DATA_BLOCK "DB104"
{ S7_Optimized_Access := 'FALSE' }
VERSION : 0.1
NON_RETAIN
   VAR
      DB104_DBD0 : Real;
      DB104_DBD4 : Real;
      DB104_DBD8 : Real;
      DB104_DBD12 : Real;
      DB104_DBD16 : Real;
      DB104_DBD20 : Real;
      DB104_DBD24 : Real;
      DB104_DBD28 : Real;
      DB104_DBD32 : Real;
      DB104_DBD36 : Real;
      DB104_DBD40 : Real;
      DB104_DBD44 : Real;
      DB104_DBD48 : Real;
      DB104_DBD52 : Real;
      DB104_DBD56 : Real;
      DB104_DBD60 : Real;
      DB104_DBD64 : Real;
      DB104_DBD68 : Real;
      DB104_DBD72 : Real;
      DB104_DBD76 : Real;
      DB104_DBD80 : Real;
      DB104_DBD84 : Real;
      DB104_DBD88 : Real;
      DB104_DBD92 : Real;
      DB104_DBD96 : Real;
      DB104_DBD100 : Real;
      DB104_DBD104 : Real;
      DB104_DBD108 : Real;
      DB104_DBD112 : Real;
      DB104_DBD116 : Real;
      DB104_DBD120 : Real;
      DB104_DBD124 : Real;
      DB104_DBD128 : Real;
      DB104_DBD132 : Real;
      DB104_DBD136 : Real;
      DB104_DBD140 : Real;
      DB104_DBD144 : Real;
      DB104_DBD148 : Real;
      DB104_DBD152 : Real;
      DB104_DBD156 : Real;
      DB104_DBD160 : Real;
      DB104_DBD164 : Real;
      DB104_DBD168 : Real;
      DB104_DBD172 : Real;
      DB104_DBD176 : Real;
      DB104_DBD180 : Real;
      DB104_DBD184 : Real;
      DB104_DBD188 : Real;
      DB104_DBD192 : Real;
      DB104_DBD196 : Real;
      DB104_DBD200 : Real;
      DB104_DBD204 : Real;
      DB104_DBD208 : Real;
      DB104_DBD212 : Real;
      DB104_DBD216 : Real;
      DB104_DBD220 : Real;
      DB104_DBD224 : Real;
      DB104_DBD228 : Real;
      DB104_DBD232 : Real;
      DB104_DBD236 : Real;
      DB104_DBD240 : Real;
      DB104_DBD244 : Real;
      DB104_DBD248 : Real;
      DB104_DBD252 : Real;
      DB104_DBD256 : Real;
      DB104_DBD260 : Real;
      DB104_DBD264 : Real;
      DB104_DBD268 : Real;
      DB104_DBD272 : Real;
      DB104_DBD276 : Real;
      DB104_DBD280 : Real;
      DB104_DBD284 : Real;
      DB104_DBD288 : Real;
      DB104_DBD292 : Real;
      DB104_DBD296 : Real;
      DB104_DBD300 : Real;
      DB104_DBD304 : Real;
      DB104_DBD308 : Real;
      DB104_DBD312 : Real;
      DB104_DBD316 : Real;
      DB104_DBD800 : Real;
      DB104_DBD804 : Real;
      DB104_DBD808 : Real;
      DB104_DBD812 : Real;
      DB104_DBD816 : Real;
      DB104_DBD820 : Real;
      DB104_DBD824 : Real;
      DB104_DBD828 : Real;
      DB104_DBD832 : Real;
      DB104_DBD836 : Real;
      DB104_DBD840 : Real;
      DB104_DBD844 : Real;
      DB104_DBD848 : Real;
      DB104_DBD852 : Real;
      DB104_DBD856 : Real;
      DB104_DBD860 : Real;
      DB104_DBD864 : Real;
      DB104_DBD868 : Real;
      DB104_DBD872 : Real;
      DB104_DBD876 : Real;
      DB104_DBD880 : Real;
      DB104_DBD884 : Real;
      DB104_DBD888 : Real;
      DB104_DBD892 : Real;
      DB104_DBD896 : Real;
      DB104_DBD900 : Real;
      DB104_DBD904 : Real;
      DB104_DBD908 : Real;
      DB104_DBD912 : Real;
      DB104_DBD916 : Real;
      DB104_DBD920 : Real;
      DB104_DBD924 : Real;
      DB104_DBD928 : Real;
      DB104_DBD932 : Real;
      DB104_DBD936 : Real;
      DB104_DBD940 : Real;
      DB104_DBD944 : Real;
      DB104_DBD948 : Real;
      DB104_DBD952 : Real;
      DB104_DBD956 : Real;
      DB104_DBD960 : Real;
      DB104_DBD964 : Real;
      DB104_DBD968 : Real;
      DB104_DBD972 : Real;
      DB104_DBD976 : Real;
      DB104_DBD980 : Real;
      DB104_DBD984 : Real;
      DB104_DBD988 : Real;
      DB104_DBD992 : Real;
      DB104_DBD996 : Real;
      DB104_DBD1000 : Real;
      DB104_DBD1004 : Real;
      DB104_DBD1008 : Real;
      DB104_DBD1012 : Real;
      DB104_DBD1016 : Real;
      DB104_DBD1020 : Real;
      DB104_DBD1024 : Real;
      DB104_DBD1028 : Real;
      DB104_DBD1032 : Real;
      DB104_DBD1036 : Real;
      DB104_DBD1040 : Real;
      DB104_DBD1044 : Real;
      DB104_DBD1048 : Real;
      DB104_DBD1052 : Real;
      DB104_DBD1056 : Real;
      DB104_DBD1060 : Real;
      DB104_DBD1064 : Real;
      DB104_DBD1068 : Real;
      DB104_DBD1072 : Real;
      DB104_DBD1076 : Real;
      DB104_DBD1080 : Real;
      DB104_DBD1084 : Real;
      DB104_DBD1088 : Real;
      DB104_DBD1092 : Real;
      DB104_DBD1096 : Real;
      DB104_DBD1100 : Real;
      DB104_DBD1104 : Real;
      DB104_DBD1108 : Real;
      DB104_DBD1112 : Real;
      DB104_DBD1116 : Real;
      DB104_DBD1600 : Real;
      DB104_DBD1604 : Real;
      DB104_DBD1608 : Real;
      DB104_DBD1612 : Real;
      DB104_DBD1616 : Real;
      DB104_DBD1620 : Real;
      DB104_DBD1624 : Real;
      DB104_DBD1628 : Real;
      DB104_DBD1632 : Real;
      DB104_DBD1636 : Real;
      DB104_DBD1640 : Real;
      DB104_DBD1644 : Real;
      DB104_DBD1648 : Real;
      DB104_DBD1652 : Real;
      DB104_DBD1656 : Real;
      DB104_DBD1660 : Real;
      DB104_DBD1664 : Real;
      DB104_DBD1668 : Real;
      DB104_DBD1672 : Real;
      DB104_DBD1676 : Real;
      DB104_DBD1680 : Real;
      DB104_DBD1684 : Real;
      DB104_DBD1688 : Real;
      DB104_DBD1692 : Real;
      DB104_DBD1696 : Real;
      DB104_DBD1700 : Real;
      DB104_DBD1704 : Real;
      DB104_DBD1708 : Real;
      DB104_DBD1712 : Real;
      DB104_DBD1716 : Real;
      DB104_DBD1720 : Real;
      DB104_DBD1724 : Real;
      DB104_DBD1728 : Real;
      DB104_DBD1732 : Real;
      DB104_DBD1736 : Real;
      DB104_DBD1740 : Real;
      DB104_DBD1744 : Real;
      DB104_DBD1748 : Real;
      DB104_DBD1752 : Real;
      DB104_DBD1756 : Real;
      DB104_DBD1760 : Real;
      DB104_DBD1764 : Real;
      DB104_DBD1768 : Real;
      DB104_DBD1772 : Real;
      DB104_DBD1776 : Real;
      DB104_DBD1780 : Real;
      DB104_DBD1784 : Real;
      DB104_DBD1788 : Real;
      DB104_DBD1792 : Real;
      DB104_DBD1796 : Real;
      DB104_DBD1800 : Real;
      DB104_DBD1804 : Real;
      DB104_DBD1808 : Real;
      DB104_DBD1812 : Real;
      DB104_DBD1816 : Real;
      DB104_DBD1820 : Real;
      DB104_DBD1824 : Real;
      DB104_DBD1828 : Real;
      DB104_DBD1832 : Real;
      DB104_DBD1836 : Real;
      DB104_DBD1840 : Real;
      DB104_DBD1844 : Real;
      DB104_DBD1848 : Real;
      DB104_DBD1852 : Real;
      DB104_DBD1856 : Real;
      DB104_DBD1860 : Real;
      DB104_DBD1864 : Real;
      DB104_DBD1868 : Real;
      DB104_DBD1872 : Real;
      DB104_DBD1876 : Real;
      DB104_DBD1880 : Real;
      DB104_DBD1884 : Real;
      DB104_DBD1888 : Real;
      DB104_DBD1892 : Real;
      DB104_DBD1896 : Real;
      DB104_DBD1900 : Real;
      DB104_DBD1904 : Real;
      DB104_DBD1908 : Real;
      DB104_DBD1912 : Real;
      DB104_DBD1916 : Real;
      DB104_DBD2400 : Real;
      DB104_DBD2404 : Real;
      DB104_DBD2408 : Real;
      DB104_DBD2412 : Real;
      DB104_DBD2416 : Real;
      DB104_DBD2420 : Real;
      DB104_DBD2424 : Real;
      DB104_DBD2428 : Real;
      DB104_DBD2432 : Real;
      DB104_DBD2436 : Real;
      DB104_DBD2440 : Real;
      DB104_DBD2444 : Real;
      DB104_DBD2448 : Real;
      DB104_DBD2452 : Real;
      DB104_DBD2456 : Real;
      DB104_DBD2460 : Real;
      DB104_DBD2464 : Real;
      DB104_DBD2468 : Real;
      DB104_DBD2472 : Real;
      DB104_DBD2476 : Real;
      DB104_DBD2480 : Real;
      DB104_DBD2484 : Real;
      DB104_DBD2488 : Real;
      DB104_DBD2492 : Real;
      DB104_DBD2496 : Real;
      DB104_DBD2500 : Real;
      DB104_DBD2504 : Real;
      DB104_DBD2508 : Real;
      DB104_DBD2512 : Real;
      DB104_DBD2516 : Real;
      DB104_DBD2520 : Real;
      DB104_DBD2524 : Real;
      DB104_DBD2528 : Real;
      DB104_DBD2532 : Real;
      DB104_DBD2536 : Real;
      DB104_DBD2540 : Real;
      DB104_DBD2544 : Real;
      DB104_DBD2548 : Real;
      DB104_DBD2552 : Real;
      DB104_DBD2556 : Real;
      DB104_DBD2560 : Real;
      DB104_DBD2564 : Real;
      DB104_DBD2568 : Real;
      DB104_DBD2572 : Real;
      DB104_DBD2576 : Real;
      DB104_DBD2580 : Real;
      DB104_DBD2584 : Real;
      DB104_DBD2588 : Real;
      DB104_DBD2592 : Real;
      DB104_DBD2596 : Real;
      DB104_DBD2600 : Real;
      DB104_DBD2604 : Real;
      DB104_DBD2608 : Real;
      DB104_DBD2612 : Real;
      DB104_DBD2616 : Real;
      DB104_DBD2620 : Real;
      DB104_DBD2624 : Real;
      DB104_DBD2628 : Real;
      DB104_DBD2632 : Real;
      DB104_DBD2636 : Real;
      DB104_DBD2640 : Real;
      DB104_DBD2644 : Real;
      DB104_DBD2648 : Real;
      DB104_DBD2652 : Real;
      DB104_DBD2656 : Real;
      DB104_DBD2660 : Real;
      DB104_DBD2664 : Real;
      DB104_DBD2668 : Real;
      DB104_DBD2672 : Real;
      DB104_DBD2676 : Real;
      DB104_DBD2680 : Real;
      DB104_DBD2684 : Real;
      DB104_DBD2688 : Real;
      DB104_DBD2692 : Real;
      DB104_DBD2696 : Real;
      DB104_DBD2700 : Real;
      DB104_DBD2704 : Real;
      DB104_DBD2708 : Real;
      DB104_DBD2712 : Real;
      DB104_DBD2716 : Real;
   END_VAR


BEGIN

END_DATA_BLOCK

DATA_BLOCK "DB101"
{ S7_Optimized_Access := 'FALSE' }
VERSION : 0.1
NON_RETAIN
   VAR
      DB101_DBW0 : Word;
      DB101_DBW2 : Word;
      DB101_DBD4 : Real;
      DB101_DBD8 : Real;
      DB101_DBD12 : Real;
      DB101_DBD16 : Real;
      DB101_DBD96 : Real;
      DB101_DBW176 : Word;
      DB101_DBW178 : Word;
      DB101_DBW180 : Word;
      DB101_DBW182 : Word;
      DB101_DBW184 : Word;
      DB101_DBW186 : Word;
      DB101_DBW188 : Word;
      DB101_DBW190 : Word;
      DB101_DBW192 : Word;
      DB101_DBW194 : Word;
      DB101_DBW196 : Word;
      DB101_DBW198 : Word;
      DB101_DBW200 : Word;
      DB101_DBW202 : Word;
      DB101_DBW204 : Word;
      DB101_DBW206 : Word;
      DB101_DBW208 : Word;
      DB101_DBW210 : Word;
      DB101_DBW212 : Word;
      DB101_DBW214 : Word;
      DB101_DBW216 : Word;
      DB101_DBW218 : Word;
      DB101_DBW220 : Word;
      DB101_DBW222 : Word;
      DB101_DBW224 : Word;
      DB101_DBW226 : Word;
      DB101_DBW228 : Word;
      DB101_DBW230 : Word;
      DB101_DBW232 : Word;
      DB101_DBW234 : Word;
      DB101_DBW236 : Word;
      DB101_DBW238 : Word;
      DB101_DBW240 : Word;
      DB101_DBW242 : Word;
      DB101_DBW244 : Word;
      DB101_DBW246 : Word;
      DB101_DBW248 : Word;
      DB101_DBW250 : Word;
      DB101_DBW252 : Word;
      DB101_DBW254 : Word;
      DB101_DBW256 : Word;
      DB101_DBW258 : Word;
      DB101_DBW260 : Word;
      DB101_DBW262 : Word;
      DB101_DBW264 : Word;
      DB101_DBW266 : Word;
      DB101_DBW268 : Word;
      DB101_DBW270 : Word;
      DB101_DBW272 : Word;
      DB101_DBW274 : Word;
      DB101_DBW276 : Word;
      DB101_DBW278 : Word;
      DB101_DBW280 : Word;
      DB101_DBW282 : Word;
      DB101_DBW284 : Word;
      DB101_DBW286 : Word;
      DB101_DBW288 : Word;
      DB101_DBW290 : Word;
      DB101_DBW292 : Word;
      DB101_DBW294 : Word;
      DB101_DBW296 : Word;
      DB101_DBW298 : Word;
      DB101_DBW300 : Word;
      DB101_DBW302 : Word;
      DB101_DBW304 : Word;
      DB101_DBW306 : Word;
      DB101_DBW308 : Word;
      DB101_DBW310 : Word;
      DB101_DBW312 : Word;
      DB101_DBW314 : Word;
      DB101_DBW316 : Word;
      DB101_DBW318 : Word;
      DB101_DBW320 : Word;
      DB101_DBW322 : Word;
      DB101_DBW324 : Word;
      DB101_DBW326 : Word;
      DB101_DBW328 : Word;
      DB101_DBW330 : Word;
      DB101_DBW332 : Word;
      DB101_DBW334 : Word;
      DB101_DBW576 : Word;
      DB101_DBW578 : Word;
      DB101_DBW580 : Word;
      DB101_DBW582 : Word;
      DB101_DBW584 : Word;
      DB101_DBW586 : Word;
      DB101_DBW588 : Word;
      DB101_DBW590 : Word;
      DB101_DBW592 : Word;
      DB101_DBW594 : Word;
      DB101_DBW596 : Word;
      DB101_DBW598 : Word;
      DB101_DBW600 : Word;
      DB101_DBW602 : Word;
      DB101_DBW604 : Word;
      DB101_DBW606 : Word;
      DB101_DBW608 : Word;
      DB101_DBW610 : Word;
      DB101_DBW612 : Word;
      DB101_DBW614 : Word;
      DB101_DBW616 : Word;
      DB101_DBW618 : Word;
      DB101_DBW620 : Word;
      DB101_DBW622 : Word;
      DB101_DBW624 : Word;
      DB101_DBW626 : Word;
      DB101_DBW628 : Word;
      DB101_DBW630 : Word;
      DB101_DBW632 : Word;
      DB101_DBW634 : Word;
      DB101_DBW636 : Word;
      DB101_DBW638 : Word;
      DB101_DBW640 : Word;
      DB101_DBW642 : Word;
      DB101_DBW644 : Word;
      DB101_DBW646 : Word;
      DB101_DBW648 : Word;
      DB101_DBW650 : Word;
      DB101_DBW652 : Word;
      DB101_DBW654 : Word;
      DB101_DBW656 : Word;
      DB101_DBW658 : Word;
      DB101_DBW660 : Word;
      DB101_DBW662 : Word;
      DB101_DBW664 : Word;
      DB101_DBW666 : Word;
      DB101_DBW668 : Word;
      DB101_DBW670 : Word;
      DB101_DBW672 : Word;
      DB101_DBW674 : Word;
      DB101_DBW676 : Word;
      DB101_DBW678 : Word;
      DB101_DBW680 : Word;
      DB101_DBW682 : Word;
      DB101_DBW684 : Word;
      DB101_DBW686 : Word;
      DB101_DBW688 : Word;
      DB101_DBW690 : Word;
      DB101_DBW692 : Word;
      DB101_DBW694 : Word;
      DB101_DBW696 : Word;
      DB101_DBW698 : Word;
      DB101_DBW700 : Word;
      DB101_DBW702 : Word;
      DB101_DBW704 : Word;
      DB101_DBW706 : Word;
      DB101_DBW708 : Word;
      DB101_DBW710 : Word;
      DB101_DBW712 : Word;
      DB101_DBW714 : Word;
      DB101_DBW716 : Word;
      DB101_DBW718 : Word;
      DB101_DBW720 : Word;
      DB101_DBW722 : Word;
      DB101_DBW724 : Word;
      DB101_DBW726 : Word;
      DB101_DBW728 : Word;
      DB101_DBW730 : Word;
      DB101_DBW732 : Word;
      DB101_DBW734 : Word;
      DB101_DBW976 : Word;
      DB101_DBW978 : Word;
      DB101_DBW980 : Word;
      DB101_DBW982 : Word;
      DB101_DBW984 : Word;
      DB101_DBW986 : Word;
      DB101_DBW988 : Word;
      DB101_DBW990 : Word;
      DB101_DBW992 : Word;
      DB101_DBW994 : Word;
      DB101_DBW1016 : Word;
      DB101_DBW1018 : Word;
      DB101_DBW1020 : Word;
      DB101_DBW1022 : Word;
      DB101_DBW1024 : Word;
      DB101_DBW1026 : Word;
      DB101_DBW1028 : Word;
      DB101_DBW1030 : Word;
      DB101_DBW1032 : Word;
      DB101_DBW1034 : Word;
      DB101_DBW1056 : Word;
      DB101_DBW1058 : Word;
      DB101_DBW1060 : Word;
      DB101_DBW1062 : Word;
      DB101_DBW1064 : Word;
      DB101_DBW1066 : Word;
      DB101_DBW1068 : Word;
      DB101_DBW1070 : Word;
      DB101_DBW1072 : Word;
      DB101_DBW1074 : Word;
      DB101_DBW1096 : Word;
      DB101_DBW1098 : Word;
      DB101_DBW1100 : Word;
      DB101_DBW1102 : Word;
      DB101_DBW1104 : Word;
      DB101_DBW1106 : Word;
      DB101_DBW1108 : Word;
      DB101_DBW1110 : Word;
      DB101_DBW1112 : Word;
      DB101_DBW1114 : Word;
      DB101_DBX1136_0 : Bool;
      DB101_DBX1136_1 : Bool;
      DB101_DBX1136_2 : Bool;
      DB101_DBX1136_3 : Bool;
      DB101_DBX1136_4 : Bool;
      DB101_DBX1136_5 : Bool;
      DB101_DBX1136_6 : Bool;
      DB101_DBX1136_7 : Bool;
      DB101_DBX1137_0 : Bool;
      DB101_DBX1137_1 : Bool;
      DB101_DBX1140_0 : Bool;
      DB101_DBX1140_1 : Bool;
      DB101_DBX1140_2 : Bool;
      DB101_DBX1140_3 : Bool;
      DB101_DBX1140_4 : Bool;
      DB101_DBX1140_5 : Bool;
      DB101_DBX1140_6 : Bool;
      DB101_DBX1140_7 : Bool;
      DB101_DBX1141_0 : Bool;
      DB101_DBX1141_1 : Bool;
      DB101_DBD1144 : Real;
      DB101_DBD1224 : Real;
      DB101_DBW1304 : Word;
      DB101_DBW1306 : Word;
      DB101_DBW1308 : Word;
      DB101_DBW1310 : Word;
      DB101_DBW1312 : Word;
      DB101_DBW1314 : Word;
      DB101_DBW1316 : Word;
      DB101_DBW1318 : Word;
      DB101_DBW1320 : Word;
      DB101_DBW1322 : Word;
      DB101_DBW1324 : Word;
      DB101_DBW1326 : Word;
      DB101_DBW1328 : Word;
      DB101_DBW1330 : Word;
      DB101_DBW1332 : Word;
      DB101_DBW1334 : Word;
      DB101_DBW1336 : Word;
      DB101_DBW1338 : Word;
      DB101_DBW1340 : Word;
      DB101_DBW1342 : Word;
      DB101_DBW1344 : Word;
      DB101_DBW1346 : Word;
      DB101_DBW1348 : Word;
      DB101_DBW1350 : Word;
      DB101_DBW1352 : Word;
      DB101_DBW1354 : Word;
      DB101_DBW1356 : Word;
      DB101_DBW1358 : Word;
      DB101_DBW1360 : Word;
      DB101_DBW1362 : Word;
      DB101_DBW1364 : Word;
      DB101_DBW1366 : Word;
      DB101_DBW1368 : Word;
      DB101_DBW1370 : Word;
      DB101_DBW1372 : Word;
      DB101_DBW1374 : Word;
      DB101_DBW1376 : Word;
      DB101_DBW1378 : Word;
      DB101_DBW1380 : Word;
      DB101_DBW1382 : Word;
      DB101_DBW1384 : Word;
      DB101_DBW1386 : Word;
      DB101_DBW1388 : Word;
      DB101_DBW1390 : Word;
      DB101_DBW1392 : Word;
      DB101_DBW1394 : Word;
      DB101_DBW1396 : Word;
      DB101_DBW1398 : Word;
      DB101_DBW1400 : Word;
      DB101_DBW1402 : Word;
      DB101_DBW1404 : Word;
      DB101_DBW1406 : Word;
      DB101_DBW1408 : Word;
      DB101_DBW1410 : Word;
      DB101_DBW1412 : Word;
      DB101_DBW1414 : Word;
      DB101_DBW1416 : Word;
      DB101_DBW1418 : Word;
      DB101_DBW1420 : Word;
      DB101_DBW1422 : Word;
      DB101_DBW1424 : Word;
      DB101_DBW1426 : Word;
      DB101_DBW1428 : Word;
      DB101_DBW1430 : Word;
      DB101_DBW1432 : Word;
      DB101_DBW1434 : Word;
      DB101_DBW1436 : Word;
      DB101_DBW1438 : Word;
      DB101_DBW1440 : Word;
      DB101_DBW1442 : Word;
      DB101_DBW1444 : Word;
      DB101_DBW1446 : Word;
      DB101_DBW1448 : Word;
      DB101_DBW1450 : Word;
      DB101_DBW1452 : Word;
      DB101_DBW1454 : Word;
      DB101_DBW1456 : Word;
      DB101_DBW1458 : Word;
      DB101_DBW1460 : Word;
      DB101_DBW1462 : Word;
      DB101_DBW1704 : Word;
      DB101_DBW1706 : Word;
      DB101_DBW1708 : Word;
      DB101_DBW1710 : Word;
      DB101_DBW1712 : Word;
      DB101_DBW1714 : Word;
      DB101_DBW1716 : Word;
      DB101_DBW1718 : Word;
      DB101_DBW1720 : Word;
      DB101_DBW1722 : Word;
      DB101_DBW1724 : Word;
      DB101_DBW1726 : Word;
      DB101_DBW1728 : Word;
      DB101_DBW1730 : Word;
      DB101_DBW1732 : Word;
      DB101_DBW1734 : Word;
      DB101_DBW1736 : Word;
      DB101_DBW1738 : Word;
      DB101_DBW1740 : Word;
      DB101_DBW1742 : Word;
      DB101_DBW1744 : Word;
      DB101_DBW1746 : Word;
      DB101_DBW1748 : Word;
      DB101_DBW1750 : Word;
      DB101_DBW1752 : Word;
      DB101_DBW1754 : Word;
      DB101_DBW1756 : Word;
      DB101_DBW1758 : Word;
      DB101_DBW1760 : Word;
      DB101_DBW1762 : Word;
      DB101_DBW1764 : Word;
      DB101_DBW1766 : Word;
      DB101_DBW1768 : Word;
      DB101_DBW1770 : Word;
      DB101_DBW1772 : Word;
      DB101_DBW1774 : Word;
      DB101_DBW1776 : Word;
      DB101_DBW1778 : Word;
      DB101_DBW1780 : Word;
      DB101_DBW1782 : Word;
      DB101_DBW1784 : Word;
      DB101_DBW1786 : Word;
      DB101_DBW1788 : Word;
      DB101_DBW1790 : Word;
      DB101_DBW1792 : Word;
      DB101_DBW1794 : Word;
      DB101_DBW1796 : Word;
      DB101_DBW1798 : Word;
      DB101_DBW1800 : Word;
      DB101_DBW1802 : Word;
      DB101_DBW1804 : Word;
      DB101_DBW1806 : Word;
      DB101_DBW1808 : Word;
      DB101_DBW1810 : Word;
      DB101_DBW1812 : Word;
      DB101_DBW1814 : Word;
      DB101_DBW1816 : Word;
      DB101_DBW1818 : Word;
      DB101_DBW1820 : Word;
      DB101_DBW1822 : Word;
      DB101_DBW1824 : Word;
      DB101_DBW1826 : Word;
      DB101_DBW1828 : Word;
      DB101_DBW1830 : Word;
      DB101_DBW1832 : Word;
      DB101_DBW1834 : Word;
      DB101_DBW1836 : Word;
      DB101_DBW1838 : Word;
      DB101_DBW1840 : Word;
      DB101_DBW1842 : Word;
      DB101_DBW1844 : Word;
      DB101_DBW1846 : Word;
      DB101_DBW1848 : Word;
      DB101_DBW1850 : Word;
      DB101_DBW1852 : Word;
      DB101_DBW1854 : Word;
      DB101_DBW1856 : Word;
      DB101_DBW1858 : Word;
      DB101_DBW1860 : Word;
      DB101_DBW1862 : Word;
      DB101_DBW2104 : Word;
      DB101_DBW2106 : Word;
      DB101_DBW2108 : Word;
      DB101_DBW2110 : Word;
      DB101_DBW2112 : Word;
      DB101_DBW2114 : Word;
      DB101_DBW2116 : Word;
      DB101_DBW2118 : Word;
      DB101_DBW2120 : Word;
      DB101_DBW2122 : Word;
      DB101_DBW2144 : Word;
      DB101_DBW2146 : Word;
      DB101_DBW2148 : Word;
      DB101_DBW2150 : Word;
      DB101_DBW2152 : Word;
      DB101_DBW2154 : Word;
      DB101_DBW2156 : Word;
      DB101_DBW2158 : Word;
      DB101_DBW2160 : Word;
      DB101_DBW2162 : Word;
      DB101_DBW2184 : Word;
      DB101_DBW2186 : Word;
      DB101_DBW2188 : Word;
      DB101_DBW2190 : Word;
      DB101_DBW2192 : Word;
      DB101_DBW2194 : Word;
      DB101_DBW2196 : Word;
      DB101_DBW2198 : Word;
      DB101_DBW2200 : Word;
      DB101_DBW2202 : Word;
      DB101_DBW2224 : Word;
      DB101_DBW2226 : Word;
      DB101_DBW2228 : Word;
      DB101_DBW2230 : Word;
      DB101_DBW2232 : Word;
      DB101_DBW2234 : Word;
      DB101_DBW2236 : Word;
      DB101_DBW2238 : Word;
      DB101_DBW2240 : Word;
      DB101_DBW2242 : Word;
      DB101_DBX2264_0 : Bool;
      DB101_DBX2264_1 : Bool;
      DB101_DBX2264_2 : Bool;
      DB101_DBX2264_3 : Bool;
      DB101_DBX2264_4 : Bool;
      DB101_DBX2264_5 : Bool;
      DB101_DBX2264_6 : Bool;
      DB101_DBX2264_7 : Bool;
      DB101_DBX2265_0 : Bool;
      DB101_DBX2265_1 : Bool;
      DB101_DBX2268_0 : Bool;
      DB101_DBX2268_1 : Bool;
      DB101_DBX2268_2 : Bool;
      DB101_DBX2268_3 : Bool;
      DB101_DBX2268_4 : Bool;
      DB101_DBX2268_5 : Bool;
      DB101_DBX2268_6 : Bool;
      DB101_DBX2268_7 : Bool;
      DB101_DBX2269_0 : Bool;
      DB101_DBX2269_1 : Bool;
      DB101_DBW2272 : Word;
      DB101_DBW2274 : Word;
      DB101_DBD2276 : Real;
      DB101_DBD2280 : Real;
      DB101_DBD2284 : Real;
      DB101_DBD2288 : Real;
      DB101_DBD2292 : Real;
      DB101_DBD2296 : Real;
      DB101_DBD2300 : Real;
      DB101_DBD2304 : Real;
      DB101_DBD2308 : Real;
      DB101_DBD2312 : Real;
      DB101_DBD2316 : Real;
      DB101_DBD2320 : Real;
      DB101_DBD2324 : Real;
      DB101_DBD2328 : Real;
      DB101_DBD2332 : Real;
      DB101_DBD2336 : Real;
      DB101_DBD2340 : Real;
      DB101_DBD2344 : Real;
      DB101_DBD2348 : Real;
      DB101_DBD2352 : Real;
      DB101_DBD2356 : Real;
      DB101_DBD2360 : Real;
      DB101_DBD2364 : Real;
      DB101_DBD2368 : Real;
      DB101_DBD2372 : Real;
      DB101_DBD2376 : Real;
      DB101_DBD2380 : Real;
      DB101_DBD2384 : Real;
      DB101_DBD2388 : Real;
      DB101_DBD2392 : Real;
      DB101_DBD2676 : Real;
      DB101_DBD2680 : Real;
      DB101_DBD2684 : Real;
      DB101_DBD2688 : Real;
      DB101_DBD2692 : Real;
      DB101_DBD2696 : Real;
      DB101_DBD2700 : Real;
      DB101_DBD2704 : Real;
      DB101_DBD2708 : Real;
      DB101_DBD2712 : Real;
      DB101_DBD2716 : Real;
      DB101_DBD2720 : Real;
      DB101_DBD2724 : Real;
      DB101_DBD2728 : Real;
      DB101_DBD2732 : Real;
      DB101_DBD2736 : Real;
      DB101_DBD2740 : Real;
      DB101_DBD2744 : Real;
      DB101_DBD2748 : Real;
      DB101_DBD2752 : Real;
      DB101_DBD2756 : Real;
      DB101_DBD2760 : Real;
      DB101_DBD2764 : Real;
      DB101_DBD2768 : Real;
      DB101_DBD2772 : Real;
      DB101_DBD2776 : Real;
      DB101_DBD2780 : Real;
      DB101_DBD2784 : Real;
      DB101_DBD2788 : Real;
      DB101_DBD2792 : Real;
      DB101_DBD3076 : Real;
      DB101_DBD3080 : Real;
      DB101_DBW3086 : Word;
      DB101_DBW3088 : Word;
      DB101_DBD3090 : Real;
      DB101_DBD3094 : Real;
      DB101_DBW3100 : Word;
      DB101_DBW3102 : Word;
      DB101_DBD3104 : Real;
      DB101_DBD3108 : Real;
      DB101_DBW3114 : Word;
      DB101_DBW3116 : Word;
      DB101_DBD3118 : Real;
      DB101_DBD3122 : Real;
      DB101_DBW3128 : Word;
      DB101_DBW3130 : Word;
      DB101_DBD3132 : Real;
      DB101_DBD3136 : Real;
      DB101_DBW3142 : Word;
      DB101_DBW3144 : Word;
      DB101_DBD3146 : Real;
      DB101_DBD3158 : Real;
      DB101_DBD3162 : Real;
      DB101_DBD3166 : Real;
      DB101_DBD3170 : Real;
      DB101_DBW3174 : Word;
      DB101_DBD3176 : Real;
      DB101_DBD3180 : Real;
      DB101_DBW3184 : Word;
      DB101_DBD3186 : Real;
      DB101_DBD3190 : Real;
      DB101_DBD3194 : Real;
      DB101_DBD3198 : Real;
      DB101_DBW3210 : Word;
      DB101_DBD3212 : Real;
      DB101_DBD3216 : Real;
      DB101_DBD3220 : Real;
      DB101_DBD3224 : Real;
      DB101_DBD3228 : Real;
      DB101_DBD3232 : Real;
      DB101_DBD3236 : Real;
      DB101_DBD3240 : Real;
      DB101_DBD3244 : Real;
      DB101_DBD3248 : Real;
      DB101_DBD3252 : Real;
      DB101_DBD3256 : Real;
      DB101_DBD3260 : Real;
      DB101_DBD3264 : Real;
      DB101_DBD3268 : Real;
      DB101_DBD3272 : Real;
      DB101_DBD3276 : Real;
      DB101_DBD3288 : Real;
      DB101_DBD3292 : Real;
      DB101_DBD3304 : Real;
      DB101_DBW3308 : Word;
      DB101_DBW3310 : Word;
      DB101_DBW3312 : Word;
      DB101_DBW3314 : Word;
      DB101_DBW3316 : Word;
      DB101_DBW3318 : Word;
      DB101_DBW3320 : Word;
      DB101_DBW3322 : Word;
      DB101_DBW3324 : Word;
      DB101_DBW3326 : Word;
      DB101_DBW3328 : Word;
      DB101_DBW3330 : Word;
      DB101_DBW3332 : Word;
      DB101_DBW3334 : Word;
      DB101_DBW3336 : Word;
      DB101_DBW3338 : Word;
      DB101_DBW3340 : Word;
      DB101_DBW3342 : Word;
      DB101_DBW3344 : Word;
      DB101_DBW3346 : Word;
      DB101_DBW3348 : Word;
      DB101_DBW3350 : Word;
      DB101_DBW3352 : Word;
      DB101_DBW3354 : Word;
      DB101_DBW3356 : Word;
      DB101_DBW3358 : Word;
      DB101_DBW3360 : Word;
      DB101_DBW3362 : Word;
      DB101_DBW3364 : Word;
      DB101_DBW3366 : Word;
      DB101_DBW3368 : Word;
      DB101_DBW3370 : Word;
      DB101_DBW3372 : Word;
      DB101_DBW3374 : Word;
      DB101_DBW3376 : Word;
      DB101_DBW3378 : Word;
      DB101_DBW3380 : Word;
      DB101_DBW3382 : Word;
      DB101_DBW3384 : Word;
      DB101_DBW3386 : Word;
      DB101_DBW3388 : Word;
      DB101_DBW3390 : Word;
      DB101_DBW3392 : Word;
      DB101_DBW3394 : Word;
      DB101_DBW3396 : Word;
      DB101_DBW3398 : Word;
      DB101_DBW3400 : Word;
      DB101_DBW3402 : Word;
      DB101_DBW3404 : Word;
      DB101_DBW3406 : Word;
      DB101_DBW3408 : Word;
      DB101_DBW3410 : Word;
      DB101_DBW3412 : Word;
      DB101_DBW3414 : Word;
      DB101_DBX3430_0 : Bool;
      DB101_DBX3430_1 : Bool;
      DB101_DBX3432_0 : Bool;
      DB101_DBW3434 : Word;
      DB101_DBW3436 : Word;
      DB101_DBW3438 : Word;
      DB101_DBW3440 : Word;
      DB101_DBW3442 : Word;
      DB101_DBW3444 : Word;
      DB101_DBW3446 : Word;
      DB101_DBW3448 : Word;
      DB101_DBW3474 : Word;
      DB101_DBW3476 : Word;
      DB101_DBW3478 : Word;
      DB101_DBW3480 : Word;
      DB101_DBW3482 : Word;
      DB101_DBW3484 : Word;
      DB101_DBW3486 : Word;
      DB101_DBW3488 : Word;
      DB101_DBW3514 : Word;
      DB101_DBW3516 : Word;
      DB101_DBW3518 : Word;
      DB101_DBW3520 : Word;
      DB101_DBW3522 : Word;
      DB101_DBW3524 : Word;
      DB101_DBW3526 : Word;
      DB101_DBW3528 : Word;
      DB101_DBW3554 : Word;
      DB101_DBW3556 : Word;
      DB101_DBW3558 : Word;
      DB101_DBW3560 : Word;
      DB101_DBW3562 : Word;
      DB101_DBW3564 : Word;
      DB101_DBW3566 : Word;
      DB101_DBW3568 : Word;
      DB101_DBD3594 : Real;
   END_VAR


BEGIN

END_DATA_BLOCK

